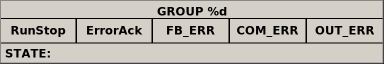
VISUALIZATION V_PH_GROUP  // 384x64
VAR_INPUT
	wIndex					:WORD;
	stSafetyStatusGroup		:ST_SAFETYStatusGroup;
	
END_VAR
    Rectangle (0,0 384x64)
    Rectangle (117,1 150x21), "GROUP %d", text variable: wIndex
    Rectangle (76,18 76x25), "ErrorAck", colour toggle: stSafetyStatusGroup.bERR_Ack
    Rectangle (152,18 77x25), "FB_ERR", colour toggle: stSafetyStatusGroup.bFB_ERR
    Rectangle (306,18 78x25), "OUT_ERR", colour toggle: stSafetyStatusGroup.bOUT_ERR
    Rectangle (229,18 77x25), "COM_ERR", colour toggle: stSafetyStatusGroup.bCOM_ERR
    Rectangle (0,18 76x25), "RunStop", colour toggle: stSafetyStatusGroup.bRUN_STOP
    Rectangle (67,44 315x19), text list: 'TL_GroupState', text index: stSafetyStatusGroup.eSAFETY_GroupState
    Label (2,44 55x19), "STATE:"
END_VISUALIZATION

(* stored: Version 1.1.0.1, ProductVersion 3.1.4024.4
   Visu V_PH_GROUP: Id {47435180-1e14-4f40-bdc0-a22139c44a3f} *)
